{attribute 'qualified_only'}


VAR_GLOBAL
END_VAR

(* stored: Version 1.1.0.1, ProductVersion 3.1.4024.12
   GVL gAlarm: Id {cd8c748c-3e37-4c83-a58a-a1c3094c1b43} *)
